Staubli VAL3: HOME.dtx

public TrajHome tTraj{}
  [home]
    frame fFrame = {fatherId=world[0]}
    num nDimension
    num nIndexFrame
    num nIndexTool
    num nZoneMove
    num nZoneType
    pointRx pO = {fatherId=world[0]}
    pointRx pPointMove = {fatherId=tTraj["home"].fFrame[0]}
    pointRx pX = {fatherId=world[0]}
    pointRx pY = {fatherId=world[0]}
    string sID = "home"
    string sProgram
    TrajJointItem tData
      [0]
        jointRx jJoint = {j1=89.750339, j2=-61.16853, j3=-123.267439, j4=-179.754871, j5=-91.659213, j6=-90.62711}
        TrajectoryItem tSuper
          [0]
            string comment
            num distance
            InstrItem iInstr[3]
              [0]
                string sData = "valve1>ON"
                string sType = "OUT"
              [1]
                string sData
                string sType
              [2]
                string sData
                string sType
            num moveType
            num nMoveId
            num nStop = 2
            num nTcpAction
            num nTime
            mdesc nom_speed = {vel=50, tmax=500, blend=off}
            bool toStop = true
